// TIA Portal project "Coffee Grinder Timer" (V17)
// Coffee Grinder Timer
// When the Start button is pressed, the grinder should run for 30s before stopping automatically.
// After stopping the buzzer will turn ON. Pressing Stop Button will turn OFF the buzzer after 5s.

(* hardware
DEVICE "S7-1200 station_1"  S7-1200 Station
   slot 0: "Rack_0"  Rack  V1.0
   slot 1: "PLC_1"  CPU 1212C AC/DC/Rly SIPLUS  6AG1 212-1BE40-4XB0  V4.5
*)

// ===== PLC "PLC_1"  CPU 1212C AC/DC/Rly SIPLUS =====

VAR_GLOBAL   // PLC tag table "Default tag table"
   "Start button" AT %I0.0 : Bool;
   "Stop button" AT %I0.1 : Bool;
   "Grinder motor" AT %Q0.0 : Bool;
   "Buzzer" AT %Q0.1 : Bool;
   "Tag_1" AT %M0.0 : Bool;
END_VAR

// folder: System blocks/Program resources

DATA_BLOCK "IEC_Timer_0_DB"   // DB1
{ S7_Optimized_Access := 'TRUE' }
AUTHOR : Simatic
FAMILY : IEC
NAME : IEC_TMR
VERSION : 1.0
// stored: InstanceOfName IEC_TIMER
"IEC_TIMER"
BEGIN
END_DATA_BLOCK

DATA_BLOCK "IEC_Timer_0_DB_1"   // DB2
{ S7_Optimized_Access := 'TRUE' }
AUTHOR : Simatic
FAMILY : IEC
NAME : IEC_TMR
VERSION : 1.0
// stored: InstanceOfName IEC_TIMER
"IEC_TIMER"
BEGIN
END_DATA_BLOCK

// folder: (top level)

ORGANIZATION_BLOCK "Main"   // OB1, LAD, ProgramCycle
TITLE = "Main Program Sweep (Cycle)"
{ S7_Optimized_Access := 'TRUE' }
VERSION : 0.1
   VAR_INPUT
      Initial_Call : Bool;   // Initial call of this OB
      Remanence : Bool;   // =True, if remanent data are available
   END_VAR
BEGIN

REGION Network 1
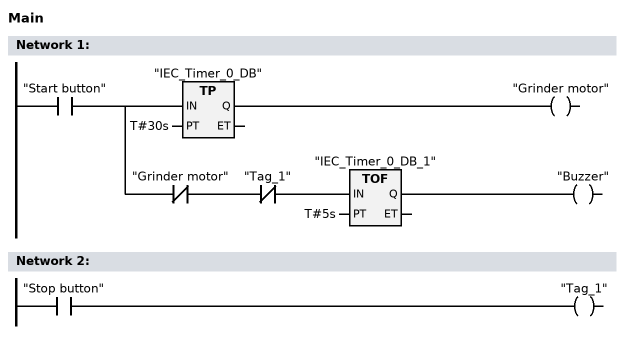
   "IEC_Timer_0_DB".TP(IN := "Start button", PT := T#30s);
   "Grinder motor" := "IEC_Timer_0_DB".Q;
   "IEC_Timer_0_DB_1".TOF(IN := "Start button" AND NOT "Grinder motor" AND NOT "Tag_1", PT := T#5s);
   "Buzzer" := "IEC_Timer_0_DB_1".Q;
END_REGION

REGION Network 2
   RUNG wire#powerrail
      Contact( "Stop button" )
      Coil( "Tag_1" )
   END_RUNG
   // the same network as SCL:
   "Tag_1" := "Stop button";
END_REGION
END_ORGANIZATION_BLOCK